{attribute addProperty BoxType "EL3201-0000-0016"}
{attribute addProperty Id "RTD_InputsAT %I*RTD_Inputs_BC62E3BB7290WcStateAT %I*WcState_F855686C1620InfoDataAT %I*InfoData_BC63D37F80100"}
{attribute addProperty CRC "830953022"}
{attribute addProperty SizeInBites "168"}
{attribute addProperty SizeInBytes "21"}
TYPE EL3201_E6230DF0 :
STRUCT
	{attribute addProperty Name "RTD_Inputs"}
	RTD_Inputs : RTD_Inputs_BC62E3BB;
	{attribute addProperty Name "WcState"}
	WcState : WcState_F855686C;
	{attribute addProperty Name "InfoData"}
	InfoData : InfoData_BC63D37F;
END_STRUCT
END_TYPE

(* stored: Version 1.2.0.0, ProductVersion 3.1.4024.9
   DUT EL3201_E6230DF0: Id {3bb28103-dccc-477d-88bf-0899a7193135} *)
